FUNCTION F_Convert10V2CO2 : INT
VAR_INPUT
	i_Value			:	INT;
END_VAR
VAR_OUTPUT
END_VAR
VAR
	r_converted2V 	: 	REAL;
	i_finalValue	:	INT;
END_VAR

// For Convertion of 0-10V Signal from 0-2000ppm

r_converted2V := i_Value * 0.061037018951994;
i_finalValue := REAL_TO_INT(r_converted2V);

F_Convert10V2CO2 := i_finalValue;

END_FUNCTION

(* stored: Version 1.1.0.1, ProductVersion 3.1.4024.4
   POU F_Convert10V2CO2: Id {981b850f-abae-4e0c-bf61-a5700408cf18}, SpecialFunc None *)
